(* CODESYS project Copy_of_Sensor_model_new.library
   TcLibraryId: TE140x Module Vendor|Copy_of_Sensor_model_new|0.0.0.3
   Company: TE140x Module Vendor
   Title: Copy_of_Sensor_model_new
   Placeholder: Copy_of_Sensor_model_new
   Version: 0.0.0.3

Project tree, tasks and I/O mapping:
  POUs/
    function block FB_Copy_of_Sensor_model_new [ST]: FB_exit, FB_init, nHResult, eInitExceptionHandling, eUpdateExceptionHandling, nExceptionCnt, stActiveException, bInitialized, bExecute
    TcCOM Wrapper/
      function block FB_Copy_of_Sensor_model_new_TcCOM_InitStruct [ST]: FB_init, FB_afterinit, Reinit, FB_exit, eObjectState, nHResult, ipTcComObject, ipADI, nTaskOid, nTaskPriority, nTaskCycleTimeNs, nTaskPort, nTaskSortOrder, eTraceLevelMax, eModuleCaller, eCallerVerification, eStepSizeAdaptation, eExecutionSequence, bExecute, eAccessLockState, eInitExceptionHandling, eUpdateExceptionHandling, stModuleBuildInfo, bInitialized, nSkippedExecutionCount, stLibraryInfo, stModuleInfo, stModuleGeneratorInfo, stSimulinkModelInfo, eCopy_of_Sensor_model_new_P_Sharing, nCopy_of_Sensor_model_new_P_Definer, stCopy_of_Sensor_model_new_P, fSimulationTime, nCycleCount, nExceptionCount, stExceptionInfo
  DUTs/
    data type ST_FB_Copy_of_Sensor_model_new_FB_Main
    data type ST_FB_Copy_of_Sensor_model_new_FB_exit
    data type ST_FB_Copy_of_Sensor_model_new_FB_init
    data type ST_GetSet_HRESULT
    data type E_FpExcptCtrlSetEx
    data type ST_GetSet_E_FpExcptCtrlSetEx
    data type ST_GetSet_ULINT
    data type ST_ExceptionInfo
    data type ST_GetSet_ST_ExceptionInfo
    data type ST_GetSet_BOOL
    data type T_matrix12xdouble
    data type T_matrix6xdouble
    data type T_matrix3xdouble
    data type E_SimTimeStep
    data type E_SolverMode
    data type E_ssMatrixType
    data type ST_RTWRTModelMethodsInfo
    data type E_slJmBdControl
    data type ST_ssSolverInfo
    data type T_matrix2xdouble
    data type ST_B_MovingAveragepitch_Copy_of_Sensor_model_new_T
    data type ST_B_MovingAveragey_Copy_of_Sensor_model_new_T
    data type ST_B_Copy_of_Sensor_model_new_T
    data type T_ZCSigState
    data type ST_PrevZCX_Copy_of_Sensor_model_new_T
    data type ST_X_Copy_of_Sensor_model_new_T
    data type ST_ExtU_Copy_of_Sensor_model_new_T
    data type ST_ExtY_Copy_of_Sensor_model_new_T
    data type ST_XDis_Copy_of_Sensor_model_new_T
    data type T_matrix2x4xdouble
    data type PLREAL
    data type T_matrix4xdoublepointer
    data type ST_ODE4_IntgData
    data type T_matrix8xuint32
    data type ST_cell_wrap_Copy_of_Sensor_model_new_T
    data type T_matrix9xdouble
    data type ST_dsp_simulink_MovingAverage_Copy_of_Sensor_model_new_T
    data type ST_DW_MovingAveragepitch_Copy_of_Sensor_model_new_T
    data type ST_DW_MovingAveragey_Copy_of_Sensor_model_new_T
    data type ST_DW_Copy_of_Sensor_model_new_T
    data type ST_x08a7a7bbd0e5d629f7d70ceec84eacfe
    data type ST_xf09845edab6c83520d8d57def6d6fe1c
    data type ST_RT_MODEL_Copy_of_Sensor_model_new_T
    data type T_matrix18xdouble
    data type ST_P_Copy_of_Sensor_model_new_T
    data type E_ModuleCaller
    data type E_CallerVerification
    data type E_StepSizeAdaptation
    data type E_ExecutionSequence1
    data type E_FpExcptCtrlSet
    data type ST_TcMatSim_ModuleGeneratorInfo
    data type ST_TcMatSim_SimulinkModelInfo
    data type E_ParameterSharingType
    data type ST_FB_Copy_of_Sensor_model_new_TcCOM_InitStruct
    data type ST_FB_Copy_of_Sensor_model_new_TcCOM_InitStruct_FB_init
    data type ST_FB_Copy_of_Sensor_model_new_TcCOM_InitStruct_FB_afterinit
    data type ST_FB_Copy_of_Sensor_model_new_TcCOM_InitStruct_Reinit
    data type ST_FB_Copy_of_Sensor_model_new_TcCOM_InitStruct_FB_Main
    data type ST_FB_Copy_of_Sensor_model_new_TcCOM_InitStruct_FB_exit
    data type ST_GetSet_TCOM_STATE
    data type ST_GetSet_ITComObject
    data type ST_GetSet_ITcADI
    data type ST_Copy_of_Sensor_model_new_U_T
    data type ST_Copy_of_Sensor_model_new_Y_T
    data type ST_Copy_of_Sensor_model_new_X_T
    data type ST_Copy_of_Sensor_model_new_DW_T
    data type ST_GetSet_OTCID
    data type ST_GetSet_UDINT
    data type ST_GetSet_UINT
    data type ST_GetSet_TcTraceLevel
    data type ST_GetSet_E_ModuleCaller
    data type ST_GetSet_E_CallerVerification
    data type ST_GetSet_E_StepSizeAdaptation
    data type ST_GetSet_E_ExecutionSequence1
    data type ST_GetSet_E_FpExcptCtrlSet
    data type ST_ModuleBuildInfo
    data type ST_GetSet_ST_ModuleBuildInfo
    data type ST_LibraryInfo
    data type ST_GetSet_ST_LibraryInfo
    data type ST_ModuleInfo
    data type ST_GetSet_ST_ModuleInfo
    data type ST_GetSet_ST_TcMatSim_ModuleGeneratorInfo
    data type ST_GetSet_ST_TcMatSim_SimulinkModelInfo
    data type ST_GetSet_E_ParameterSharingType
    data type ST_GetSet_ST_P_Copy_of_Sensor_model_new_T
    data type ST_GetSet_LREAL
  Version/
    global variables Global_Version
*)

// DUTs/ST_FB_Copy_of_Sensor_model_new_FB_Main
{attribute 'TcIecLibraryType'}
{attribute 'hide'}
TYPE ST_FB_Copy_of_Sensor_model_new_FB_Main : 
	STRUCT
		{attribute 'GUID' := '18071995-0000-0000-0000-000000000018'}
		pInst : PVOID;
		result : BOOL;
		 {attribute 'hide'}
		_reserved1 : UINT_24_56;
	END_STRUCT
END_TYPE

// DUTs/ST_FB_Copy_of_Sensor_model_new_FB_exit
{attribute 'TcIecLibraryType'}
{attribute 'hide'}
TYPE ST_FB_Copy_of_Sensor_model_new_FB_exit : 
	STRUCT
		{attribute 'GUID' := '18071995-0000-0000-0000-000000000018'}
		pInst : PVOID;
		bInCopyCode : BOOL;
		result : BOOL;
		 {attribute 'hide'}
		_reserved1 : UINT_16_48;
	END_STRUCT
END_TYPE

// DUTs/ST_FB_Copy_of_Sensor_model_new_FB_init
{attribute 'TcIecLibraryType'}
{attribute 'hide'}
TYPE ST_FB_Copy_of_Sensor_model_new_FB_init : 
	STRUCT
		{attribute 'GUID' := '18071995-0000-0000-0000-000000000018'}
		pInst : PVOID;
		bInitRetains : BOOL;
		bInCopyCode : BOOL;
		result : BOOL;
		 {attribute 'hide'}
		_reserved1 : UINT_8_40;
	END_STRUCT
END_TYPE

// DUTs/ST_GetSet_HRESULT
{attribute 'TcIecLibraryType'}
{attribute 'hide'}
TYPE ST_GetSet_HRESULT : 
	STRUCT
		{attribute 'GUID' := '18071995-0000-0000-0000-000000000018'}
		pInst : PVOID;
		{attribute 'GUID' := '18071995-0000-0000-0000-000000000019'}
		nParam : HRESULT;
		 {attribute 'hide'}
		_reserved1 : UINT_0_32;
	END_STRUCT
END_TYPE

// DUTs/E_FpExcptCtrlSetEx
(* Generated from type 'TcMgSdk.FpExcptCtrlSetEx' *)
{attribute 'TcIecLibraryType'}
TYPE E_FpExcptCtrlSetEx : (
	CallerExceptions:=1, 	(* Use the floating point exception settings provided by the caller *)
	ThrowExceptions:=3, 	(* Enable floating point exceptions on invalid operations and divisions by zero *)
	SuppressExceptions:=13, 	(* Disable floating point exceptions. *)
	LogExceptions:=19, 	(* Log exception information. *)
	LogAndHold:=51, 	(* Log exception information and puase execution of the cyclic code after completion of the actual cycle *)
	LogAndCatch:=83, 	(* Log exception information and immediately terminate execution of the cyclic code. Reinitialization is required to restart. *)
	LogAndDump:=147, 	(* Log exception information, create a dump file with detailed exception information and try to continue execution of the cyclic code *)
	LogHoldAndDump:=179, 	(* Log exception information, create a dump file with detailed exception information and puase execution of the cyclic code after completion of the actual cycle *)
	LogCatchAndDump:=211	(* Log exception information, create a dump file with detailed exception information and immediately terminate execution of the cyclic code. Reinitialization is required to restart. *)
) USINT;
END_TYPE

// DUTs/ST_GetSet_E_FpExcptCtrlSetEx
{attribute 'TcIecLibraryType'}
{attribute 'hide'}
TYPE ST_GetSet_E_FpExcptCtrlSetEx : 
	STRUCT
		{attribute 'GUID' := '18071995-0000-0000-0000-000000000018'}
		pInst : PVOID;
		eParam : E_FpExcptCtrlSetEx;
		 {attribute 'hide'}
		_reserved1 : UINT_24_56;
	END_STRUCT
END_TYPE

// DUTs/ST_GetSet_ULINT
{attribute 'TcIecLibraryType'}
{attribute 'hide'}
TYPE ST_GetSet_ULINT : 
	STRUCT
		{attribute 'GUID' := '18071995-0000-0000-0000-000000000018'}
		pInst : PVOID;
		nParam : ULINT;
	END_STRUCT
END_TYPE

// DUTs/ST_ExceptionInfo
(* Generated from type 'TcMgSdk.ExceptionInfo' *)
{attribute 'TcIecLibraryType'}
TYPE ST_ExceptionInfo : 
	STRUCT
		(* Generated from item 'ExceptionCode' *)
		nExceptionCode : DINT;
		(* Generated from item 'TmxName' *)
		{attribute 'GUID' := '18071995-0000-0000-0000-00010000007F'}
		sTmxName : STRING(127);
		(* Generated from item 'TmxVersion' *)
		nTmxVersion : ARRAY [0..3] OF UDINT;
		(* Generated from item 'InstructionAddr' *)
		nInstructionAddr : UDINT;
		(* Generated from item 'ReturnAddr' *)
		nReturnAddr : ARRAY [0..3] OF UDINT;
		(* Generated from item 'DumpCreated' *)
		bDumpCreated : BOOL;
		 {attribute 'hide'}
		_reserved1 : ARRAY [1..3] OF USINT;
	END_STRUCT
END_TYPE

// DUTs/ST_GetSet_ST_ExceptionInfo
{attribute 'TcIecLibraryType'}
{attribute 'hide'}
TYPE ST_GetSet_ST_ExceptionInfo : 
	STRUCT
		{attribute 'GUID' := '18071995-0000-0000-0000-000000000018'}
		pInst : PVOID;
		stParam : ST_ExceptionInfo;
		 {attribute 'hide'}
		_reserved1 : UINT_0_32;
	END_STRUCT
END_TYPE

// DUTs/ST_GetSet_BOOL
{attribute 'TcIecLibraryType'}
{attribute 'hide'}
TYPE ST_GetSet_BOOL : 
	STRUCT
		{attribute 'GUID' := '18071995-0000-0000-0000-000000000018'}
		pInst : PVOID;
		bParam : BOOL;
		 {attribute 'hide'}
		_reserved1 : UINT_24_56;
	END_STRUCT
END_TYPE

// DUTs/T_matrix12xdouble
(* Generated from type 'matrix12xdouble' *)
{attribute 'TcIecLibraryType'}
TYPE T_matrix12xdouble : ARRAY [0..11] OF LREAL;
END_TYPE

// DUTs/T_matrix6xdouble
(* Generated from type 'matrix6xdouble' *)
{attribute 'TcIecLibraryType'}
TYPE T_matrix6xdouble : ARRAY [0..5] OF LREAL;
END_TYPE

// DUTs/T_matrix3xdouble
(* Generated from type 'matrix3xdouble' *)
{attribute 'TcIecLibraryType'}
TYPE T_matrix3xdouble : ARRAY [0..2] OF LREAL;
END_TYPE

// DUTs/E_SimTimeStep
(* Generated from type 'SimTimeStep' *)
{attribute 'TcIecLibraryType'}
{attribute 'qualified_only' := 'true'}
TYPE E_SimTimeStep : (MINOR_TIME_STEP:=0, MAJOR_TIME_STEP:=1) DINT;
END_TYPE

// DUTs/E_SolverMode
(* Generated from type 'SolverMode' *)
{attribute 'TcIecLibraryType'}
{attribute 'qualified_only' := 'true'}
TYPE E_SolverMode : (SOLVER_MODE_AUTO:=0, SOLVER_MODE_SINGLETASKING:=1, SOLVER_MODE_MULTITASKING:=2) DINT;
END_TYPE

// DUTs/E_ssMatrixType
(* Generated from type 'ssMatrixType' *)
{attribute 'TcIecLibraryType'}
{attribute 'qualified_only' := 'true'}
TYPE E_ssMatrixType : (SS_MATRIX_NONE:=0, SS_MATRIX_CONSTANT:=1, SS_MATRIX_TIMEDEP:=2, SS_MATRIX_STATEDEP:=3) DINT;
END_TYPE

// DUTs/ST_RTWRTModelMethodsInfo
(* Generated from type 'RTWRTModelMethodsInfo' *)
{attribute 'TcIecLibraryType'}
TYPE ST_RTWRTModelMethodsInfo : 
	STRUCT
		(* Generated from item 'rtModelPtr' *)
		{attribute 'GUID' := '18071995-0000-0000-0000-000000000018'}
		prtModelPtr : PVOID;
		(* Generated from item 'rtmInitSizesFcn' *)
		{attribute 'GUID' := '18071995-0000-0000-0000-000000000018'}
		prtmInitSizesFcn : PVOID;
		(* Generated from item 'rtmInitSampTimesFcn' *)
		{attribute 'GUID' := '18071995-0000-0000-0000-000000000018'}
		prtmInitSampTimesFcn : PVOID;
		(* Generated from item 'rtmStartFcn' *)
		{attribute 'GUID' := '18071995-0000-0000-0000-000000000018'}
		prtmStartFcn : PVOID;
		(* Generated from item 'rtmOutputsFcn' *)
		{attribute 'GUID' := '18071995-0000-0000-0000-000000000018'}
		prtmOutputsFcn : PVOID;
		(* Generated from item 'rtmUpdateFcn' *)
		{attribute 'GUID' := '18071995-0000-0000-0000-000000000018'}
		prtmUpdateFcn : PVOID;
		(* Generated from item 'rtmDervisFcn' *)
		{attribute 'GUID' := '18071995-0000-0000-0000-000000000018'}
		prtmDervisFcn : PVOID;
		(* Generated from item 'rtmProjectionFcn' *)
		{attribute 'GUID' := '18071995-0000-0000-0000-000000000018'}
		prtmProjectionFcn : PVOID;
		(* Generated from item 'rtmMassMatrixFcn' *)
		{attribute 'GUID' := '18071995-0000-0000-0000-000000000018'}
		prtmMassMatrixFcn : PVOID;
		(* Generated from item 'rtmForcingFunctionFcn' *)
		{attribute 'GUID' := '18071995-0000-0000-0000-000000000018'}
		prtmForcingFunctionFcn : PVOID;
		(* Generated from item 'rtmTerminateFcn' *)
		{attribute 'GUID' := '18071995-0000-0000-0000-000000000018'}
		prtmTerminateFcn : PVOID;
		(* Generated from item 'rtmDiscreteEventsFcn' *)
		{attribute 'GUID' := '18071995-0000-0000-0000-000000000018'}
		prtmDiscreteEventsFcn : PVOID;
	END_STRUCT
END_TYPE

// DUTs/E_slJmBdControl
(* Generated from type 'slJmBdControl' *)
{attribute 'TcIecLibraryType'}
{attribute 'qualified_only' := 'true'}
TYPE E_slJmBdControl : (SL_JM_BD_AUTO:=0, SL_JM_BD_SPARSE_PERTURBATION:=1, SL_JM_BD_FULL_PERTURBATION:=2, SL_JM_BD_SPARSE_ANALYTICAL:=3, SL_JM_BD_FULL_ANALYTICAL:=4) DINT;
END_TYPE

// DUTs/ST_ssSolverInfo
(* Generated from type 'ssSolverInfo' *)
{attribute 'TcIecLibraryType'}
TYPE ST_ssSolverInfo : 
	STRUCT
		(* Generated from item 'rtModelPtr' *)
		{attribute 'GUID' := '18071995-0000-0000-0000-000000000018'}
		prtModelPtr : PVOID;
		simTimeStepPtr : POINTER TO E_SimTimeStep;
		(* Generated from item 'solverData' *)
		{attribute 'GUID' := '18071995-0000-0000-0000-000000000018'}
		psolverData : PVOID;
		solverName : POINTER TO SINT;
		(* Generated from item 'isVariableStepSolver' *)
		bisVariableStepSolver : BOOL;
		(* Generated from item 'solverNeedsReset' *)
		bsolverNeedsReset : BOOL;
		 {attribute 'hide'}
		_reserved1 : UINT;
		(* Generated from item 'solverMode' *)
		esolverMode : E_SolverMode;
		(* Generated from item 'solverStopTime' *)
		fsolverStopTime : LREAL;
		stepSizePtr : POINTER TO LREAL;
		(* Generated from item 'minStepSize' *)
		fminStepSize : LREAL;
		(* Generated from item 'maxStepSize' *)
		fmaxStepSize : LREAL;
		(* Generated from item 'fixedStepSize' *)
		ffixedStepSize : LREAL;
		(* Generated from item 'solverShapePreserveControl' *)
		nsolverShapePreserveControl : DINT;
		(* Generated from item 'solverMaxConsecutiveMinStep' *)
		nsolverMaxConsecutiveMinStep : DINT;
		(* Generated from item 'maxNumMinSteps' *)
		nmaxNumMinSteps : DINT;
		(* Generated from item 'solverMaxOrder' *)
		nsolverMaxOrder : DINT;
		(* Generated from item 'solverConsecutiveZCsStepRelTol' *)
		fsolverConsecutiveZCsStepRelTol : LREAL;
		(* Generated from item 'solverMaxConsecutiveZCs' *)
		nsolverMaxConsecutiveZCs : DINT;
		(* Generated from item 'solverExtrapolationOrder' *)
		nsolverExtrapolationOrder : DINT;
		(* Generated from item 'solverNumberNewtonIterations' *)
		nsolverNumberNewtonIterations : DINT;
		(* Generated from item 'solverRefineFactor' *)
		nsolverRefineFactor : DINT;
		(* Generated from item 'solverRelTol' *)
		fsolverRelTol : LREAL;
		(* Generated from item 'unused_real_T_1' *)
		funused_real_T_1 : LREAL;
		dXPtr : POINTER TO POINTER TO LREAL;
		tPtr : POINTER TO POINTER TO LREAL;
		numContStatesPtr : POINTER TO DINT;
		contStatesPtr : POINTER TO POINTER TO LREAL;
		numPeriodicContStatesPtr : POINTER TO DINT;
		periodicContStateIndicesPtr : POINTER TO POINTER TO DINT;
		periodicContStateRangesPtr : POINTER TO POINTER TO LREAL;
		zcSignalVector : POINTER TO LREAL;
		zcEventsVector : POINTER TO USINT;
		zcSignalAttrib : POINTER TO USINT;
		(* Generated from item 'zcSignalVectorLength' *)
		nzcSignalVectorLength : DINT;
		 {attribute 'hide'}
		_reserved2 : UINT_0_32;
		reserved : POINTER TO USINT;
		(* Generated from item 'foundContZcEvents' *)
		bfoundContZcEvents : BOOL;
		(* Generated from item 'isAtLeftPostOfContZcEvent' *)
		bisAtLeftPostOfContZcEvent : BOOL;
		(* Generated from item 'isAtRightPostOfContZcEvent' *)
		bisAtRightPostOfContZcEvent : BOOL;
		(* Generated from item 'adaptiveZcDetection' *)
		badaptiveZcDetection : BOOL;
		(* Generated from item 'numZcSignals' *)
		nnumZcSignals : DINT;
		(* Generated from item 'stateProjection' *)
		bstateProjection : BOOL;
		(* Generated from item 'robustResetMethod' *)
		brobustResetMethod : BOOL;
		(* Generated from item 'updateJacobianAtReset' *)
		bupdateJacobianAtReset : BOOL;
		(* Generated from item 'consistencyChecking' *)
		bconsistencyChecking : BOOL;
		(* Generated from item 'massMatrixType' *)
		emassMatrixType : E_ssMatrixType;
		(* Generated from item 'massMatrixNzMax' *)
		nmassMatrixNzMax : DINT;
		 {attribute 'hide'}
		_reserved3 : UINT_0_32;
		massMatrixIr : POINTER TO DINT;
		massMatrixJc : POINTER TO DINT;
		massMatrixPr : POINTER TO LREAL;
		errStatusPtr : POINTER TO POINTER TO SINT;
		modelMethodsPtr : POINTER TO ST_RTWRTModelMethodsInfo;
		(* Generated from item 'zcThreshold' *)
		fzcThreshold : LREAL;
		(* Generated from item 'reserved_1' *)
		nreserved_1 : DINT;
		(* Generated from item 'consecutiveZCsError' *)
		nconsecutiveZCsError : DINT;
		(* Generated from item 'CTOutputIncnstWithState' *)
		bCTOutputIncnstWithState : BOOL;
		(* Generated from item 'isComputingJacobian' *)
		bisComputingJacobian : BOOL;
		 {attribute 'hide'}
		_reserved4 : UINT;
		(* Generated from item 'solverJacobianMethodControl' *)
		esolverJacobianMethodControl : E_slJmBdControl;
		(* Generated from item 'ignoredZcDiagnostic' *)
		nignoredZcDiagnostic : DINT;
		(* Generated from item 'maskedZcDiagnostic' *)
		nmaskedZcDiagnostic : DINT;
		(* Generated from item 'isOutputMethodComputed' *)
		bisOutputMethodComputed : BOOL;
		 {attribute 'hide'}
		_reserved5 : ARRAY [1..3] OF USINT;
		(* Generated from item 'maxZcBracketingIterations' *)
		nmaxZcBracketingIterations : DINT;
		(* Generated from item 'isMinorTimeStepWithModeChange' *)
		bisMinorTimeStepWithModeChange : BOOL;
		 {attribute 'hide'}
		_reserved6 : ARRAY [1..3] OF USINT;
		(* Generated from item 'maxZcPerStep' *)
		nmaxZcPerStep : DINT;
		zcSignalPtr : POINTER TO POINTER TO LREAL;
		(* Generated from item 'contStateDisabledPtr' *)
		bcontStateDisabledPtr : POINTER TO POINTER TO BOOL;
		(* Generated from item 'isContModeFrozen' *)
		bisContModeFrozen : BOOL;
		 {attribute 'hide'}
		_reserved7 : ARRAY [1..7] OF USINT;
	END_STRUCT
END_TYPE

// DUTs/T_matrix2xdouble
(* Generated from type 'matrix2xdouble' *)
{attribute 'TcIecLibraryType'}
TYPE T_matrix2xdouble : ARRAY [0..1] OF LREAL;
END_TYPE

// DUTs/ST_B_MovingAveragepitch_Copy_of_Sensor_model_new_T
(* Generated from type 'B_MovingAveragepitch_Copy_of_Sensor_model_new_T' *)
{attribute 'TcIecLibraryType'}
TYPE ST_B_MovingAveragepitch_Copy_of_Sensor_model_new_T : 
	STRUCT
		(* Generated from item 'MovingAveragepitch' *)
		fMovingAveragepitch : LREAL;
	END_STRUCT
END_TYPE

// DUTs/ST_B_MovingAveragey_Copy_of_Sensor_model_new_T
(* Generated from type 'B_MovingAveragey_Copy_of_Sensor_model_new_T' *)
{attribute 'TcIecLibraryType'}
TYPE ST_B_MovingAveragey_Copy_of_Sensor_model_new_T : 
	STRUCT
		(* Generated from item 'MovingAveragey' *)
		fMovingAveragey : LREAL;
	END_STRUCT
END_TYPE

// DUTs/ST_B_Copy_of_Sensor_model_new_T
(* Generated from type 'B_Copy_of_Sensor_model_new_T' *)
{attribute 'TcIecLibraryType'}
TYPE ST_B_Copy_of_Sensor_model_new_T : 
	STRUCT
		(* Generated from item 'UnitDelay' *)
		fUnitDelay : LREAL;
		(* Generated from item 'UnitDelay1' *)
		fUnitDelay1 : LREAL;
		(* Generated from item 'Convert_to_meters' *)
		aConvert_to_meters : T_matrix12xdouble;
		(* Generated from item 'z' *)
		fz : LREAL;
		(* Generated from item 'roll' *)
		froll : LREAL;
		(* Generated from item 'pitch' *)
		fpitch : LREAL;
		(* Generated from item 'offset_airgaps' *)
		aoffset_airgaps : T_matrix6xdouble;
		(* Generated from item 'corrected_airgaps' *)
		acorrected_airgaps : T_matrix12xdouble;
		(* Generated from item 'n_vertical_sensors_rejected' *)
		fn_vertical_sensors_rejected : LREAL;
		(* Generated from item 'n_lateral_sensors_rejected' *)
		fn_lateral_sensors_rejected : LREAL;
		(* Generated from item 'trigger_vertical_filter' *)
		ftrigger_vertical_filter : LREAL;
		(* Generated from item 'trigger_lateral_filter' *)
		ftrigger_lateral_filter : LREAL;
		(* Generated from item 'y' *)
		fy : LREAL;
		(* Generated from item 'yaw' *)
		fyaw : LREAL;
		(* Generated from item 'offset_airgaps_c' *)
		aoffset_airgaps_c : T_matrix6xdouble;
		(* Generated from item 'airgap_nominal_ems' *)
		aairgap_nominal_ems : T_matrix3xdouble;
		(* Generated from item 'Switch' *)
		aSwitch : T_matrix3xdouble;
		(* Generated from item 'Switch1' *)
		aSwitch1 : T_matrix2xdouble;
		(* Generated from item 'Integrator1' *)
		fIntegrator1 : LREAL;
		(* Generated from item 'RelationalOperator1' *)
		bRelationalOperator1 : BOOL;
		 {attribute 'hide'}
		_reserved1 : ARRAY [1..7] OF USINT;
		(* Generated from item 'MovingAveragez' *)
		stMovingAveragez : ST_B_MovingAveragepitch_Copy_of_Sensor_model_new_T;
		(* Generated from item 'MovingAverageyaw' *)
		stMovingAverageyaw : ST_B_MovingAveragey_Copy_of_Sensor_model_new_T;
		(* Generated from item 'MovingAveragey' *)
		stMovingAveragey : ST_B_MovingAveragey_Copy_of_Sensor_model_new_T;
		(* Generated from item 'MovingAverageroll' *)
		stMovingAverageroll : ST_B_MovingAveragepitch_Copy_of_Sensor_model_new_T;
		(* Generated from item 'MovingAveragepitch' *)
		stMovingAveragepitch : ST_B_MovingAveragepitch_Copy_of_Sensor_model_new_T;
	END_STRUCT
END_TYPE

// DUTs/T_ZCSigState
(* Generated from type 'ZCSigState' *)
{attribute 'TcIecLibraryType'}
TYPE T_ZCSigState : USINT;
END_TYPE

// DUTs/ST_PrevZCX_Copy_of_Sensor_model_new_T
(* Generated from type 'PrevZCX_Copy_of_Sensor_model_new_T' *)
{attribute 'TcIecLibraryType'}
TYPE ST_PrevZCX_Copy_of_Sensor_model_new_T : 
	STRUCT
		(* Generated from item 'Integrator_Reset_ZCE' *)
		nIntegrator_Reset_ZCE : T_ZCSigState;
		(* Generated from item 'Integrator1_Reset_ZCE' *)
		nIntegrator1_Reset_ZCE : T_ZCSigState;
	END_STRUCT
END_TYPE

// DUTs/ST_X_Copy_of_Sensor_model_new_T
(* Generated from type 'X_Copy_of_Sensor_model_new_T' *)
{attribute 'TcIecLibraryType'}
TYPE ST_X_Copy_of_Sensor_model_new_T : 
	STRUCT
		(* Generated from item 'Integrator_CSTATE' *)
		fIntegrator_CSTATE : LREAL;
		(* Generated from item 'Integrator1_CSTATE' *)
		fIntegrator1_CSTATE : LREAL;
	END_STRUCT
END_TYPE

// DUTs/ST_ExtU_Copy_of_Sensor_model_new_T
(* Generated from type 'ExtU_Copy_of_Sensor_model_new_T' *)
{attribute 'TcIecLibraryType'}
TYPE ST_ExtU_Copy_of_Sensor_model_new_T : 
	STRUCT
		(* Generated from item 'Newsensorairgaps' *)
		aNewsensorairgaps : T_matrix12xdouble;
	END_STRUCT
END_TYPE

// DUTs/ST_ExtY_Copy_of_Sensor_model_new_T
(* Generated from type 'ExtY_Copy_of_Sensor_model_new_T' *)
{attribute 'TcIecLibraryType'}
TYPE ST_ExtY_Copy_of_Sensor_model_new_T : 
	STRUCT
		(* Generated from item 'z_filtered' *)
		fz_filtered : LREAL;
		(* Generated from item 'roll_filtered' *)
		froll_filtered : LREAL;
		(* Generated from item 'pitch_filtered' *)
		fpitch_filtered : LREAL;
		(* Generated from item 'y_filtered' *)
		fy_filtered : LREAL;
		(* Generated from item 'yaw_filtered' *)
		fyaw_filtered : LREAL;
		(* Generated from item 'offset_airgaps' *)
		aoffset_airgaps : T_matrix6xdouble;
		(* Generated from item 'offset_airgaps_ems' *)
		aoffset_airgaps_ems : T_matrix6xdouble;
		(* Generated from item 'n_vertical_sensors_rejected' *)
		fn_vertical_sensors_rejected : LREAL;
		(* Generated from item 'n_lateral_sensors_rejected' *)
		fn_lateral_sensors_rejected : LREAL;
		(* Generated from item 'z' *)
		fz : LREAL;
		(* Generated from item 'roll' *)
		froll : LREAL;
		(* Generated from item 'pitch' *)
		fpitch : LREAL;
		(* Generated from item 'y' *)
		fy : LREAL;
		(* Generated from item 'yaw' *)
		fyaw : LREAL;
		(* Generated from item 'airgap_nominal_ems' *)
		aairgap_nominal_ems : T_matrix3xdouble;
	END_STRUCT
END_TYPE

// DUTs/ST_XDis_Copy_of_Sensor_model_new_T
(* Generated from type 'XDis_Copy_of_Sensor_model_new_T' *)
{attribute 'TcIecLibraryType'}
TYPE ST_XDis_Copy_of_Sensor_model_new_T : 
	STRUCT
		(* Generated from item 'Integrator_CSTATE' *)
		bIntegrator_CSTATE : BOOL;
		(* Generated from item 'Integrator1_CSTATE' *)
		bIntegrator1_CSTATE : BOOL;
	END_STRUCT
END_TYPE

// DUTs/T_matrix2x4xdouble
(* Generated from type 'matrix2x4xdouble' *)
{attribute 'TcIecLibraryType'}
TYPE T_matrix2x4xdouble : ARRAY [0..3,0..1] OF LREAL;
END_TYPE

// DUTs/PLREAL
{attribute 'TcIecLibraryType'}
TYPE PLREAL : POINTER TO LREAL;
END_TYPE

// DUTs/T_matrix4xdoublepointer
(* Generated from type 'matrix4xdouble *' *)
{attribute 'TcIecLibraryType'}
{attribute 'BaseTypeGUID' := '2CE33DB5-EBD3-49F7-1FA0-F8105FFA7B54'}
TYPE T_matrix4xdoublepointer : ARRAY [0..3] OF PLREAL;
END_TYPE

// DUTs/ST_ODE4_IntgData
(* Generated from type 'ODE4_IntgData' *)
{attribute 'TcIecLibraryType'}
{attribute 'pack_mode' := '1'}
TYPE ST_ODE4_IntgData : 
	STRUCT
		y : POINTER TO LREAL;
		(* Generated from item 'f' *)
		af : T_matrix4xdoublepointer;
	END_STRUCT
END_TYPE

// DUTs/T_matrix8xuint32
(* Generated from type 'matrix8xuint32' *)
{attribute 'TcIecLibraryType'}
TYPE T_matrix8xuint32 : ARRAY [0..7] OF UDINT;
END_TYPE

// DUTs/ST_cell_wrap_Copy_of_Sensor_model_new_T
(* Generated from type 'cell_wrap_Copy_of_Sensor_model_new_T' *)
{attribute 'TcIecLibraryType'}
TYPE ST_cell_wrap_Copy_of_Sensor_model_new_T : 
	STRUCT
		(* Generated from item 'f1' *)
		af1 : T_matrix8xuint32;
	END_STRUCT
END_TYPE

// DUTs/T_matrix9xdouble
(* Generated from type 'matrix9xdouble' *)
{attribute 'TcIecLibraryType'}
TYPE T_matrix9xdouble : ARRAY [0..8] OF LREAL;
END_TYPE

// DUTs/ST_dsp_simulink_MovingAverage_Copy_of_Sensor_model_new_T
(* Generated from type 'dsp_simulink_MovingAverage_Copy_of_Sensor_model_new_T' *)
{attribute 'TcIecLibraryType'}
TYPE ST_dsp_simulink_MovingAverage_Copy_of_Sensor_model_new_T : 
	STRUCT
		(* Generated from item 'matlabCodegenIsDeleted' *)
		bmatlabCodegenIsDeleted : BOOL;
		 {attribute 'hide'}
		_reserved1 : ARRAY [1..3] OF USINT;
		(* Generated from item 'isInitialized' *)
		nisInitialized : DINT;
		(* Generated from item 'isSetupComplete' *)
		bisSetupComplete : BOOL;
		(* Generated from item 'TunablePropsChanged' *)
		bTunablePropsChanged : BOOL;
		 {attribute 'hide'}
		_reserved2 : UINT;
		(* Generated from item 'inputVarSize' *)
		stinputVarSize : ST_cell_wrap_Copy_of_Sensor_model_new_T;
		(* Generated from item 'NumChannels' *)
		nNumChannels : DINT;
		(* Generated from item 'FrameLength' *)
		nFrameLength : DINT;
		 {attribute 'hide'}
		_reserved3 : UDINT;
		(* Generated from item 'pCumSum' *)
		fpCumSum : LREAL;
		(* Generated from item 'pCumSumRev' *)
		apCumSumRev : T_matrix9xdouble;
		(* Generated from item 'pCumRevIndex' *)
		fpCumRevIndex : LREAL;
		(* Generated from item 'pModValueRev' *)
		fpModValueRev : LREAL;
	END_STRUCT
END_TYPE

// DUTs/ST_DW_MovingAveragepitch_Copy_of_Sensor_model_new_T
(* Generated from type 'DW_MovingAveragepitch_Copy_of_Sensor_model_new_T' *)
{attribute 'TcIecLibraryType'}
TYPE ST_DW_MovingAveragepitch_Copy_of_Sensor_model_new_T : 
	STRUCT
		(* Generated from item 'obj' *)
		stobj : ST_dsp_simulink_MovingAverage_Copy_of_Sensor_model_new_T;
		(* Generated from item 'objisempty' *)
		bobjisempty : BOOL;
		 {attribute 'hide'}
		_reserved1 : ARRAY [1..7] OF USINT;
	END_STRUCT
END_TYPE

// DUTs/ST_DW_MovingAveragey_Copy_of_Sensor_model_new_T
(* Generated from type 'DW_MovingAveragey_Copy_of_Sensor_model_new_T' *)
{attribute 'TcIecLibraryType'}
TYPE ST_DW_MovingAveragey_Copy_of_Sensor_model_new_T : 
	STRUCT
		(* Generated from item 'obj' *)
		stobj : ST_dsp_simulink_MovingAverage_Copy_of_Sensor_model_new_T;
		(* Generated from item 'objisempty' *)
		bobjisempty : BOOL;
		 {attribute 'hide'}
		_reserved1 : ARRAY [1..7] OF USINT;
	END_STRUCT
END_TYPE

// DUTs/ST_DW_Copy_of_Sensor_model_new_T
(* Generated from type 'DW_Copy_of_Sensor_model_new_T' *)
{attribute 'TcIecLibraryType'}
TYPE ST_DW_Copy_of_Sensor_model_new_T : 
	STRUCT
		(* Generated from item 'UnitDelay_DSTATE' *)
		fUnitDelay_DSTATE : LREAL;
		(* Generated from item 'UnitDelay1_DSTATE' *)
		fUnitDelay1_DSTATE : LREAL;
		(* Generated from item 'MovingAveragez' *)
		stMovingAveragez : ST_DW_MovingAveragepitch_Copy_of_Sensor_model_new_T;
		(* Generated from item 'MovingAverageyaw' *)
		stMovingAverageyaw : ST_DW_MovingAveragey_Copy_of_Sensor_model_new_T;
		(* Generated from item 'MovingAveragey' *)
		stMovingAveragey : ST_DW_MovingAveragey_Copy_of_Sensor_model_new_T;
		(* Generated from item 'MovingAverageroll' *)
		stMovingAverageroll : ST_DW_MovingAveragepitch_Copy_of_Sensor_model_new_T;
		(* Generated from item 'MovingAveragepitch' *)
		stMovingAveragepitch : ST_DW_MovingAveragepitch_Copy_of_Sensor_model_new_T;
	END_STRUCT
END_TYPE

// DUTs/ST_x08a7a7bbd0e5d629f7d70ceec84eacfe
(* Generated from type 'x08a7a7bbd0e5d629f7d70ceec84eacfe' *)
{attribute 'TcIecLibraryType'}
TYPE ST_x08a7a7bbd0e5d629f7d70ceec84eacfe : 
	STRUCT
		(* Generated from item 'numContStates' *)
		nnumContStates : DINT;
		(* Generated from item 'numPeriodicContStates' *)
		nnumPeriodicContStates : DINT;
		(* Generated from item 'numSampTimes' *)
		nnumSampTimes : DINT;
	END_STRUCT
END_TYPE

// DUTs/ST_xf09845edab6c83520d8d57def6d6fe1c
(* Generated from type 'xf09845edab6c83520d8d57def6d6fe1c' *)
{attribute 'TcIecLibraryType'}
TYPE ST_xf09845edab6c83520d8d57def6d6fe1c : 
	STRUCT
		(* Generated from item 'clockTick0' *)
		nclockTick0 : UDINT;
		(* Generated from item 'clockTickH0' *)
		nclockTickH0 : UDINT;
		(* Generated from item 'stepSize0' *)
		fstepSize0 : LREAL;
		(* Generated from item 'clockTick1' *)
		nclockTick1 : UDINT;
		(* Generated from item 'clockTickH1' *)
		nclockTickH1 : UDINT;
		(* Generated from item 'tStart' *)
		ftStart : LREAL;
		(* Generated from item 'simTimeStep' *)
		esimTimeStep : E_SimTimeStep;
		(* Generated from item 'stopRequestedFlag' *)
		bstopRequestedFlag : BOOL;
		 {attribute 'hide'}
		_reserved1 : ARRAY [1..3] OF USINT;
		t : POINTER TO LREAL;
		(* Generated from item 'tArray' *)
		atArray : T_matrix2xdouble;
	END_STRUCT
END_TYPE

// DUTs/ST_RT_MODEL_Copy_of_Sensor_model_new_T
(* Generated from type 'RT_MODEL_Copy_of_Sensor_model_new_T' *)
{attribute 'TcIecLibraryType'}
{attribute 'pack_mode' := '1'}
TYPE ST_RT_MODEL_Copy_of_Sensor_model_new_T : 
	STRUCT
		errorStatus : POINTER TO SINT;
		solverInfo : POINTER TO ST_ssSolverInfo;
		blockIO : POINTER TO ST_B_Copy_of_Sensor_model_new_T;
		prevZCSigState : POINTER TO ST_PrevZCX_Copy_of_Sensor_model_new_T;
		contStates : POINTER TO ST_X_Copy_of_Sensor_model_new_T;
		periodicContStateIndices : POINTER TO DINT;
		periodicContStateRanges : POINTER TO LREAL;
		derivs : POINTER TO LREAL;
		inputs : POINTER TO ST_ExtU_Copy_of_Sensor_model_new_T;
		outputs : POINTER TO ST_ExtY_Copy_of_Sensor_model_new_T;
		contStateDisabled : POINTER TO ST_XDis_Copy_of_Sensor_model_new_T;
		(* Generated from item 'zCCacheNeedsReset' *)
		bzCCacheNeedsReset : BOOL;
		(* Generated from item 'derivCacheNeedsReset' *)
		bderivCacheNeedsReset : BOOL;
		(* Generated from item 'CTOutputIncnstWithState' *)
		bCTOutputIncnstWithState : BOOL;
		 {attribute 'hide'}
		_reserved1 : UINT_8_40;
		(* Generated from item 'odeY' *)
		aodeY : T_matrix2xdouble;
		(* Generated from item 'odeF' *)
		aodeF : T_matrix2x4xdouble;
		(* Generated from item 'intgData' *)
		stintgData : ST_ODE4_IntgData;
		dwork : POINTER TO ST_DW_Copy_of_Sensor_model_new_T;
		(* Generated from item 'Sizes' *)
		stSizes : ST_x08a7a7bbd0e5d629f7d70ceec84eacfe;
		 {attribute 'hide'}
		_reserved2 : UDINT;
		(* Generated from item 'Timing' *)
		stTiming : ST_xf09845edab6c83520d8d57def6d6fe1c;
	END_STRUCT
END_TYPE

// DUTs/T_matrix18xdouble
(* Generated from type 'matrix18xdouble' *)
{attribute 'TcIecLibraryType'}
TYPE T_matrix18xdouble : ARRAY [0..17] OF LREAL;
END_TYPE

// DUTs/ST_P_Copy_of_Sensor_model_new_T
(* Generated from type 'P_Copy_of_Sensor_model_new_T' *)
{attribute 'TcIecLibraryType'}
TYPE ST_P_Copy_of_Sensor_model_new_T : 
	STRUCT
		(* Generated from item 'Laser_magnet_offset_EMS' *)
		aLaser_magnet_offset_EMS : T_matrix6xdouble;
		(* Generated from item 'Laser_magnet_offset_HEMS' *)
		aLaser_magnet_offset_HEMS : T_matrix6xdouble;
		(* Generated from item 'coords_lat_sensors' *)
		acoords_lat_sensors : T_matrix12xdouble;
		(* Generated from item 'coords_vert_sensors' *)
		acoords_vert_sensors : T_matrix18xdouble;
		(* Generated from item 'cycle_time' *)
		fcycle_time : LREAL;
		(* Generated from item 'lateral_filter_window_cycles' *)
		flateral_filter_window_cycles : LREAL;
		(* Generated from item 'n_sensors_v' *)
		fn_sensors_v : LREAL;
		(* Generated from item 'vertical_filter_window_cycles' *)
		fvertical_filter_window_cycles : LREAL;
		(* Generated from item 'z_com' *)
		fz_com : LREAL;
		(* Generated from item 'UnitDelay_InitialCondition' *)
		fUnitDelay_InitialCondition : LREAL;
		(* Generated from item 'UnitDelay1_InitialCondition' *)
		fUnitDelay1_InitialCondition : LREAL;
		(* Generated from item 'Convert_to_meters_Gain' *)
		fConvert_to_meters_Gain : LREAL;
		(* Generated from item 'Integrator_IC' *)
		fIntegrator_IC : LREAL;
		(* Generated from item 'Integrator1_IC' *)
		fIntegrator1_IC : LREAL;
		(* Generated from item 'Constant_Value' *)
		fConstant_Value : LREAL;
	END_STRUCT
END_TYPE

// DUTs/E_ModuleCaller
(* Generated from type 'TcMgSdk.ModuleCaller' *)
{attribute 'TcIecLibraryType'}
TYPE E_ModuleCaller : (
	CyclicTask:=0, 	(* Add to the specified cyclic caller tasks. *)
	Module:=1	(* Don't add to cyclic callers. The module can be called from other TwinCAT modules (e. g. a PLC). *)
) DINT;
END_TYPE

// DUTs/E_CallerVerification
(* Generated from type 'TcMgSdk.CallerVerification' *)
{attribute 'TcIecLibraryType'}
TYPE E_CallerVerification : (
	Default:=0, 	(* Verify the caller task only if the "ModuleCaller" parameter is set to "Module" but not when added to cyclic caller tasks. *)
	Always:=1, 	(* Always verify the caller context to prevent concurrent execution of model code and corresponding DataArea mappings. *)
	Never:=2	(* Skip caller verification to reduce execution times. *)
) DINT;
END_TYPE

// DUTs/E_StepSizeAdaptation
(* Generated from type 'TcMgSdk.StepSizeAdaptation' *)
{attribute 'TcIecLibraryType'}
TYPE E_StepSizeAdaptation : (
	RequireMatchingTaskCycleTime:=0, 	(* Don't accept task cycle times other than the Simulink step sizes. *)
	UseTaskCycleTime:=1, 	(* Adapt the Smulink step sizes to the task cycle times. *)
	UseModelStepSize:=2	(* Keep the Smulink step sizes, independent of the callers cycle time. *)
) DINT;
END_TYPE

// DUTs/E_ExecutionSequence1
(* Generated from type 'TcMgSdk.ExecutionSequence1' *)
{attribute 'TcIecLibraryType'}
TYPE E_ExecutionSequence1 : (
	UpdateBeforeOutputMapping:=0, 	(* Input mapping -> State and output update -> Output mapping -> ADS processing *)
	IoAtTaskBegin:=1	(* Input mapping -> Code execution -> Output update -> ADS processing *)
) DINT;
END_TYPE

// DUTs/E_FpExcptCtrlSet
(* Generated from type 'TcMgSdk.FpExcptCtrlSet' *)
{attribute 'TcIecLibraryType'}
TYPE E_FpExcptCtrlSet : (
	CallerExceptions:=1, 	(* Use the floating point exception settings provided by the caller *)
	ThrowExceptions:=3, 	(* Enable floating point exceptions on invalid operations and divisions by zero *)
	SuppressExceptions:=5	(* Disable floating point exceptions. *)
) USINT;
END_TYPE

// DUTs/ST_TcMatSim_ModuleGeneratorInfo
(* Generated from type 'TcMatSim.ModuleGeneratorInfo' *)
{attribute 'TcIecLibraryType'}
TYPE ST_TcMatSim_ModuleGeneratorInfo : 
	STRUCT
		(* Generated from item 'MatlabVersion' *)
		nMatlabVersion : ARRAY [0..3] OF UDINT;
		(* Generated from item 'TE140xVersion' *)
		nTE140xVersion : ARRAY [0..3] OF UDINT;
	END_STRUCT
END_TYPE

// DUTs/ST_TcMatSim_SimulinkModelInfo
(* Generated from type 'TcMatSim.SimulinkModelInfo' *)
{attribute 'TcIecLibraryType'}
TYPE ST_TcMatSim_SimulinkModelInfo : 
	STRUCT
		(* Generated from item 'ModelName' *)
		{attribute 'GUID' := '18071995-0000-0000-0000-00010000007F'}
		sModelName : STRING(127);
		(* Generated from item 'SimulinkVersion' *)
		nSimulinkVersion : ARRAY [0..3] OF UDINT;
		(* Generated from item 'ModelVersion' *)
		nModelVersion : ARRAY [0..3] OF UDINT;
		(* Generated from item 'ModelChecksum' *)
		nModelChecksum : ARRAY [0..3] OF UDINT;
	END_STRUCT
END_TYPE

// DUTs/E_ParameterSharingType
(* Generated from type 'ParameterSharingType' *)
{attribute 'TcIecLibraryType'}
TYPE E_ParameterSharingType : (
	Define:=0, 	(* This module instance defines the parameter values for all further instances of this module class. Exactly one instance of this module class must use this option. *)
	Inherit:=1	(* This module instance inherits the parameter values from the instance of this module class configured to "Define" the parameter values. Model parameters configured at this instsance are ignored. *)
) DINT;
END_TYPE

// DUTs/ST_FB_Copy_of_Sensor_model_new_TcCOM_InitStruct
{attribute 'TcIecLibraryType'}
TYPE ST_FB_Copy_of_Sensor_model_new_TcCOM_InitStruct : 
	STRUCT
		{attribute 'GUID' := '18071995-0000-0000-0000-000000000061'}
		eObjState : TCOM_STATE := TCOM_STATE.TCOM_STATE_OP;
		{attribute 'GUID' := '18071995-0000-0000-0000-00010000007F'}
		sObjName : STRING(127);
		{attribute 'GUID' := '18071995-0000-0000-0000-00000000000F'}
		nOid : OTCID := 4294967295;
		{attribute 'GUID' := '18071995-0000-0000-0000-00000000000F'}
		nTaskOid : OTCID;
		nTaskSortOrder : UDINT;
		{attribute 'GUID' := '8007AE3B-86BB-40F2-B385-EF87FCC239A4'}
		eTraceLevelMax : TcTraceLevel := TcTraceLevel.tlInfo;
		eModuleCaller : E_ModuleCaller := E_ModuleCaller.CyclicTask;
		eCallerVerification : E_CallerVerification := E_CallerVerification.Default;
		eStepSizeAdaptation : E_StepSizeAdaptation := E_StepSizeAdaptation.RequireMatchingTaskCycleTime;
		eExecutionSequence : E_ExecutionSequence1 := E_ExecutionSequence1.UpdateBeforeOutputMapping;
		bExecute : BOOL := TRUE;
		 {attribute 'hide'}
		_reserved1 : ARRAY [1..3] OF USINT;
		{attribute 'GUID' := '18071995-0000-0000-0000-000000000061'}
		eAccessLockState : TCOM_STATE := TCOM_STATE.TCOM_STATE_OP;
		eInitExceptionHandling : E_FpExcptCtrlSet := E_FpExcptCtrlSet.CallerExceptions;
		eUpdateExceptionHandling : E_FpExcptCtrlSetEx := E_FpExcptCtrlSetEx.CallerExceptions;
		 {attribute 'hide'}
		_reserved2 : UINT;
		stModuleGeneratorInfo : ST_TcMatSim_ModuleGeneratorInfo;
		stSimulinkModelInfo : ST_TcMatSim_SimulinkModelInfo;
		eCopy_of_Sensor_model_new_P_Sharing : E_ParameterSharingType := E_ParameterSharingType.Define;
		 {attribute 'hide'}
		_reserved3 : UDINT;
		stCopy_of_Sensor_model_new_P : ST_P_Copy_of_Sensor_model_new_T := (aLaser_magnet_offset_EMS := [0.028731,0.0309094,0.02935319,0.02708477,0.02997081,0.02840083], aLaser_magnet_offset_HEMS := [0.01781551,0.01975221,0.02068667,0.02088624,0.01921297,0.0207209], acoords_lat_sensors := [0.8879802,0.0045598,0.8879802,0.0045598,0.0147302,0.0045598,0.0147302,0.0045598,-0.8585198,0.0045598,-0.8585198,0.0045598], acoords_vert_sensors := [0.8879802,0.3635598,0.0,0.8879802,-0.3544402,0.0,0.1997302,0.3785598,0.0,-0.1702698,-0.3694402,0.0,-0.8585198,0.3635598,0.0,-0.8585198,-0.3544402,0.0], fcycle_time := 0.0015, flateral_filter_window_cycles := 10, fn_sensors_v := 6, fvertical_filter_window_cycles := 10, fz_com := 0.5706599999999999, fUnitDelay_InitialCondition := 0, fUnitDelay1_InitialCondition := 0, fConvert_to_meters_Gain := 0.001, fIntegrator_IC := 0, fIntegrator1_IC := 0, fConstant_Value := 1);
	END_STRUCT
END_TYPE

// DUTs/ST_FB_Copy_of_Sensor_model_new_TcCOM_InitStruct_FB_init
{attribute 'TcIecLibraryType'}
{attribute 'hide'}
TYPE ST_FB_Copy_of_Sensor_model_new_TcCOM_InitStruct_FB_init : 
	STRUCT
		{attribute 'GUID' := '18071995-0000-0000-0000-000000000018'}
		pInst : PVOID;
		bInitRetains : BOOL;
		bInCopyCode : BOOL;
		 {attribute 'hide'}
		_reserved1 : UINT_16_48;
		stInit : REFERENCE TO ST_FB_Copy_of_Sensor_model_new_TcCOM_InitStruct;
		result : BOOL;
		 {attribute 'hide'}
		_reserved2 : UINT_24_56;
	END_STRUCT
END_TYPE

// DUTs/ST_FB_Copy_of_Sensor_model_new_TcCOM_InitStruct_FB_afterinit
{attribute 'TcIecLibraryType'}
{attribute 'hide'}
TYPE ST_FB_Copy_of_Sensor_model_new_TcCOM_InitStruct_FB_afterinit : 
	STRUCT
		{attribute 'GUID' := '18071995-0000-0000-0000-000000000018'}
		pInst : PVOID;
		result : BOOL;
		 {attribute 'hide'}
		_reserved1 : UINT_24_56;
	END_STRUCT
END_TYPE

// DUTs/ST_FB_Copy_of_Sensor_model_new_TcCOM_InitStruct_Reinit
{attribute 'TcIecLibraryType'}
{attribute 'hide'}
TYPE ST_FB_Copy_of_Sensor_model_new_TcCOM_InitStruct_Reinit : 
	STRUCT
		{attribute 'GUID' := '18071995-0000-0000-0000-000000000018'}
		pInst : PVOID;
		stReInit : ST_FB_Copy_of_Sensor_model_new_TcCOM_InitStruct;
		result : BOOL;
		 {attribute 'hide'}
		_reserved1 : ARRAY [1..7] OF USINT;
	END_STRUCT
END_TYPE

// DUTs/ST_FB_Copy_of_Sensor_model_new_TcCOM_InitStruct_FB_Main
{attribute 'TcIecLibraryType'}
{attribute 'hide'}
TYPE ST_FB_Copy_of_Sensor_model_new_TcCOM_InitStruct_FB_Main : 
	STRUCT
		{attribute 'GUID' := '18071995-0000-0000-0000-000000000018'}
		pInst : PVOID;
		result : BOOL;
		 {attribute 'hide'}
		_reserved1 : UINT_24_56;
	END_STRUCT
END_TYPE

// DUTs/ST_FB_Copy_of_Sensor_model_new_TcCOM_InitStruct_FB_exit
{attribute 'TcIecLibraryType'}
{attribute 'hide'}
TYPE ST_FB_Copy_of_Sensor_model_new_TcCOM_InitStruct_FB_exit : 
	STRUCT
		{attribute 'GUID' := '18071995-0000-0000-0000-000000000018'}
		pInst : PVOID;
		bInCopyCode : BOOL;
		result : BOOL;
		 {attribute 'hide'}
		_reserved1 : UINT_16_48;
	END_STRUCT
END_TYPE

// DUTs/ST_GetSet_TCOM_STATE
{attribute 'TcIecLibraryType'}
{attribute 'hide'}
TYPE ST_GetSet_TCOM_STATE : 
	STRUCT
		{attribute 'GUID' := '18071995-0000-0000-0000-000000000018'}
		pInst : PVOID;
		{attribute 'GUID' := '18071995-0000-0000-0000-000000000061'}
		eParam : TCOM_STATE;
		 {attribute 'hide'}
		_reserved1 : UINT_0_32;
	END_STRUCT
END_TYPE

// DUTs/ST_GetSet_ITComObject
{attribute 'TcIecLibraryType'}
{attribute 'hide'}
TYPE ST_GetSet_ITComObject : 
	STRUCT
		{attribute 'GUID' := '18071995-0000-0000-0000-000000000018'}
		pInst : PVOID;
		{attribute 'GUID' := '00000012-0000-0000-E000-000000000064'}
		ipParam : ITComObject;
	END_STRUCT
END_TYPE

// DUTs/ST_GetSet_ITcADI
{attribute 'TcIecLibraryType'}
{attribute 'hide'}
TYPE ST_GetSet_ITcADI : 
	STRUCT
		{attribute 'GUID' := '18071995-0000-0000-0000-000000000018'}
		pInst : PVOID;
		{attribute 'GUID' := '03000012-0000-0000-E000-000000000064'}
		ipParam : ITcADI;
	END_STRUCT
END_TYPE

// DUTs/ST_Copy_of_Sensor_model_new_U_T
(* Generated from type 'Copy_of_Sensor_model_new_U_T' *)
{attribute 'TcIecLibraryType'}
TYPE ST_Copy_of_Sensor_model_new_U_T : 
	STRUCT
		(* Generated from item 'Newsensorairgaps' *)
		aNewsensorairgaps : T_matrix12xdouble;
	END_STRUCT
END_TYPE

// DUTs/ST_Copy_of_Sensor_model_new_Y_T
(* Generated from type 'Copy_of_Sensor_model_new_Y_T' *)
{attribute 'TcIecLibraryType'}
TYPE ST_Copy_of_Sensor_model_new_Y_T : 
	STRUCT
		(* Generated from item 'z_filtered' *)
		fz_filtered : LREAL;
		(* Generated from item 'roll_filtered' *)
		froll_filtered : LREAL;
		(* Generated from item 'pitch_filtered' *)
		fpitch_filtered : LREAL;
		(* Generated from item 'y_filtered' *)
		fy_filtered : LREAL;
		(* Generated from item 'yaw_filtered' *)
		fyaw_filtered : LREAL;
		(* Generated from item 'offset_airgaps' *)
		aoffset_airgaps : T_matrix6xdouble;
		(* Generated from item 'offset_airgaps_ems' *)
		aoffset_airgaps_ems : T_matrix6xdouble;
		(* Generated from item 'n_vertical_sensors_rejected' *)
		fn_vertical_sensors_rejected : LREAL;
		(* Generated from item 'n_lateral_sensors_rejected' *)
		fn_lateral_sensors_rejected : LREAL;
		(* Generated from item 'z' *)
		fz : LREAL;
		(* Generated from item 'roll' *)
		froll : LREAL;
		(* Generated from item 'pitch' *)
		fpitch : LREAL;
		(* Generated from item 'y' *)
		fy : LREAL;
		(* Generated from item 'yaw' *)
		fyaw : LREAL;
		(* Generated from item 'airgap_nominal_ems' *)
		aairgap_nominal_ems : T_matrix3xdouble;
	END_STRUCT
END_TYPE

// DUTs/ST_Copy_of_Sensor_model_new_X_T
(* Generated from type 'Copy_of_Sensor_model_new_X_T' *)
{attribute 'TcIecLibraryType'}
TYPE ST_Copy_of_Sensor_model_new_X_T : 
	STRUCT
		(* Generated from item 'Integrator_CSTATE' *)
		fIntegrator_CSTATE : LREAL;
		(* Generated from item 'Integrator1_CSTATE' *)
		fIntegrator1_CSTATE : LREAL;
	END_STRUCT
END_TYPE

// DUTs/ST_Copy_of_Sensor_model_new_DW_T
(* Generated from type 'Copy_of_Sensor_model_new_DW_T' *)
{attribute 'TcIecLibraryType'}
TYPE ST_Copy_of_Sensor_model_new_DW_T : 
	STRUCT
		(* Generated from item 'UnitDelay_DSTATE' *)
		fUnitDelay_DSTATE : LREAL;
		(* Generated from item 'UnitDelay1_DSTATE' *)
		fUnitDelay1_DSTATE : LREAL;
		(* Generated from item 'MovingAveragez' *)
		stMovingAveragez : ST_DW_MovingAveragepitch_Copy_of_Sensor_model_new_T;
		(* Generated from item 'MovingAverageyaw' *)
		stMovingAverageyaw : ST_DW_MovingAveragey_Copy_of_Sensor_model_new_T;
		(* Generated from item 'MovingAveragey' *)
		stMovingAveragey : ST_DW_MovingAveragey_Copy_of_Sensor_model_new_T;
		(* Generated from item 'MovingAverageroll' *)
		stMovingAverageroll : ST_DW_MovingAveragepitch_Copy_of_Sensor_model_new_T;
		(* Generated from item 'MovingAveragepitch' *)
		stMovingAveragepitch : ST_DW_MovingAveragepitch_Copy_of_Sensor_model_new_T;
	END_STRUCT
END_TYPE

// DUTs/ST_GetSet_OTCID
{attribute 'TcIecLibraryType'}
{attribute 'hide'}
TYPE ST_GetSet_OTCID : 
	STRUCT
		{attribute 'GUID' := '18071995-0000-0000-0000-000000000018'}
		pInst : PVOID;
		{attribute 'GUID' := '18071995-0000-0000-0000-00000000000F'}
		nParam : OTCID;
		 {attribute 'hide'}
		_reserved1 : UINT_0_32;
	END_STRUCT
END_TYPE

// DUTs/ST_GetSet_UDINT
{attribute 'TcIecLibraryType'}
{attribute 'hide'}
TYPE ST_GetSet_UDINT : 
	STRUCT
		{attribute 'GUID' := '18071995-0000-0000-0000-000000000018'}
		pInst : PVOID;
		nParam : UDINT;
		 {attribute 'hide'}
		_reserved1 : UINT_0_32;
	END_STRUCT
END_TYPE

// DUTs/ST_GetSet_UINT
{attribute 'TcIecLibraryType'}
{attribute 'hide'}
TYPE ST_GetSet_UINT : 
	STRUCT
		{attribute 'GUID' := '18071995-0000-0000-0000-000000000018'}
		pInst : PVOID;
		nParam : UINT;
		 {attribute 'hide'}
		_reserved1 : UINT_16_48;
	END_STRUCT
END_TYPE

// DUTs/ST_GetSet_TcTraceLevel
{attribute 'TcIecLibraryType'}
{attribute 'hide'}
TYPE ST_GetSet_TcTraceLevel : 
	STRUCT
		{attribute 'GUID' := '18071995-0000-0000-0000-000000000018'}
		pInst : PVOID;
		{attribute 'GUID' := '8007AE3B-86BB-40F2-B385-EF87FCC239A4'}
		eParam : TcTraceLevel;
		 {attribute 'hide'}
		_reserved1 : UINT_0_32;
	END_STRUCT
END_TYPE

// DUTs/ST_GetSet_E_ModuleCaller
{attribute 'TcIecLibraryType'}
{attribute 'hide'}
TYPE ST_GetSet_E_ModuleCaller : 
	STRUCT
		{attribute 'GUID' := '18071995-0000-0000-0000-000000000018'}
		pInst : PVOID;
		eParam : E_ModuleCaller;
		 {attribute 'hide'}
		_reserved1 : UINT_0_32;
	END_STRUCT
END_TYPE

// DUTs/ST_GetSet_E_CallerVerification
{attribute 'TcIecLibraryType'}
{attribute 'hide'}
TYPE ST_GetSet_E_CallerVerification : 
	STRUCT
		{attribute 'GUID' := '18071995-0000-0000-0000-000000000018'}
		pInst : PVOID;
		eParam : E_CallerVerification;
		 {attribute 'hide'}
		_reserved1 : UINT_0_32;
	END_STRUCT
END_TYPE

// DUTs/ST_GetSet_E_StepSizeAdaptation
{attribute 'TcIecLibraryType'}
{attribute 'hide'}
TYPE ST_GetSet_E_StepSizeAdaptation : 
	STRUCT
		{attribute 'GUID' := '18071995-0000-0000-0000-000000000018'}
		pInst : PVOID;
		eParam : E_StepSizeAdaptation;
		 {attribute 'hide'}
		_reserved1 : UINT_0_32;
	END_STRUCT
END_TYPE

// DUTs/ST_GetSet_E_ExecutionSequence1
{attribute 'TcIecLibraryType'}
{attribute 'hide'}
TYPE ST_GetSet_E_ExecutionSequence1 : 
	STRUCT
		{attribute 'GUID' := '18071995-0000-0000-0000-000000000018'}
		pInst : PVOID;
		eParam : E_ExecutionSequence1;
		 {attribute 'hide'}
		_reserved1 : UINT_0_32;
	END_STRUCT
END_TYPE

// DUTs/ST_GetSet_E_FpExcptCtrlSet
{attribute 'TcIecLibraryType'}
{attribute 'hide'}
TYPE ST_GetSet_E_FpExcptCtrlSet : 
	STRUCT
		{attribute 'GUID' := '18071995-0000-0000-0000-000000000018'}
		pInst : PVOID;
		eParam : E_FpExcptCtrlSet;
		 {attribute 'hide'}
		_reserved1 : UINT_24_56;
	END_STRUCT
END_TYPE

// DUTs/ST_ModuleBuildInfo
(* Generated from type 'TcMgSdk.ModuleBuildInfo' *)
{attribute 'TcIecLibraryType'}
TYPE ST_ModuleBuildInfo : 
	STRUCT
		(* Generated from item 'TcBuild' *)
		nTcBuild : UDINT;
		(* Generated from item 'TcRevision' *)
		nTcRevision : UDINT;
		(* Generated from item 'Debug' *)
		bDebug : BOOL;
		 {attribute 'hide'}
		_reserved1 : ARRAY [1..3] OF USINT;
	END_STRUCT
END_TYPE

// DUTs/ST_GetSet_ST_ModuleBuildInfo
{attribute 'TcIecLibraryType'}
{attribute 'hide'}
TYPE ST_GetSet_ST_ModuleBuildInfo : 
	STRUCT
		{attribute 'GUID' := '18071995-0000-0000-0000-000000000018'}
		pInst : PVOID;
		stParam : ST_ModuleBuildInfo;
		 {attribute 'hide'}
		_reserved1 : UINT_0_32;
	END_STRUCT
END_TYPE

// DUTs/ST_LibraryInfo
(* Generated from type 'TcMgSdk.LibraryInfo' *)
{attribute 'TcIecLibraryType'}
TYPE ST_LibraryInfo : 
	STRUCT
		(* Generated from item 'FileVersion' *)
		nFileVersion : ARRAY [0..3] OF UDINT;
		(* Generated from item 'ProductVersion' *)
		nProductVersion : ARRAY [0..3] OF UDINT;
		(* Generated from item 'VendorName' *)
		{attribute 'GUID' := '18071995-0000-0000-0000-00010000007F'}
		sVendorName : STRING(127);
		(* Generated from item 'LibraryName' *)
		{attribute 'GUID' := '18071995-0000-0000-0000-00010000007F'}
		sLibraryName : STRING(127);
		(* Generated from item 'LibraryVersion' *)
		nLibraryVersion : ARRAY [0..3] OF UDINT;
		(* Generated from item 'LibraryId' *)
		{attribute 'GUID' := '18071995-0000-0000-0000-00010000007F'}
		sLibraryId : STRING(127);
		(* Generated from item 'LibraryGUID' *)
		{attribute 'GUID' := '18071995-0000-0000-0000-000000000024'}
		nLibraryGUID : CLSID;
		(* Generated from item 'TcSdkVersion' *)
		nTcSdkVersion : ARRAY [0..3] OF UDINT;
		(* Generated from item 'Compiler' *)
		{attribute 'GUID' := '18071995-0000-0000-0000-00010000007F'}
		sCompiler : STRING(127);
		(* Generated from item 'Debug' *)
		bDebug : BOOL;
		 {attribute 'hide'}
		_reserved1 : ARRAY [1..7] OF USINT;
	END_STRUCT
END_TYPE

// DUTs/ST_GetSet_ST_LibraryInfo
{attribute 'TcIecLibraryType'}
{attribute 'hide'}
TYPE ST_GetSet_ST_LibraryInfo : 
	STRUCT
		{attribute 'GUID' := '18071995-0000-0000-0000-000000000018'}
		pInst : PVOID;
		stParam : ST_LibraryInfo;
	END_STRUCT
END_TYPE

// DUTs/ST_ModuleInfo
(* Generated from type 'TcMgSdk.ModuleInfo' *)
{attribute 'TcIecLibraryType'}
TYPE ST_ModuleInfo : 
	STRUCT
		(* Generated from item 'ClassName' *)
		{attribute 'GUID' := '18071995-0000-0000-0000-00010000007F'}
		sClassName : STRING(127);
		(* Generated from item 'CommonClassId' *)
		{attribute 'GUID' := '18071995-0000-0000-0000-000000000024'}
		nCommonClassId : CLSID;
		(* Generated from item 'VersionClassId' *)
		{attribute 'GUID' := '18071995-0000-0000-0000-000000000024'}
		nVersionClassId : CLSID;
	END_STRUCT
END_TYPE

// DUTs/ST_GetSet_ST_ModuleInfo
{attribute 'TcIecLibraryType'}
{attribute 'hide'}
TYPE ST_GetSet_ST_ModuleInfo : 
	STRUCT
		{attribute 'GUID' := '18071995-0000-0000-0000-000000000018'}
		pInst : PVOID;
		stParam : ST_ModuleInfo;
	END_STRUCT
END_TYPE

// DUTs/ST_GetSet_ST_TcMatSim_ModuleGeneratorInfo
{attribute 'TcIecLibraryType'}
{attribute 'hide'}
TYPE ST_GetSet_ST_TcMatSim_ModuleGeneratorInfo : 
	STRUCT
		{attribute 'GUID' := '18071995-0000-0000-0000-000000000018'}
		pInst : PVOID;
		stParam : ST_TcMatSim_ModuleGeneratorInfo;
	END_STRUCT
END_TYPE

// DUTs/ST_GetSet_ST_TcMatSim_SimulinkModelInfo
{attribute 'TcIecLibraryType'}
{attribute 'hide'}
TYPE ST_GetSet_ST_TcMatSim_SimulinkModelInfo : 
	STRUCT
		{attribute 'GUID' := '18071995-0000-0000-0000-000000000018'}
		pInst : PVOID;
		stParam : ST_TcMatSim_SimulinkModelInfo;
	END_STRUCT
END_TYPE

// DUTs/ST_GetSet_E_ParameterSharingType
{attribute 'TcIecLibraryType'}
{attribute 'hide'}
TYPE ST_GetSet_E_ParameterSharingType : 
	STRUCT
		{attribute 'GUID' := '18071995-0000-0000-0000-000000000018'}
		pInst : PVOID;
		eParam : E_ParameterSharingType;
		 {attribute 'hide'}
		_reserved1 : UINT_0_32;
	END_STRUCT
END_TYPE

// DUTs/ST_GetSet_ST_P_Copy_of_Sensor_model_new_T
{attribute 'TcIecLibraryType'}
{attribute 'hide'}
TYPE ST_GetSet_ST_P_Copy_of_Sensor_model_new_T : 
	STRUCT
		{attribute 'GUID' := '18071995-0000-0000-0000-000000000018'}
		pInst : PVOID;
		stParam : ST_P_Copy_of_Sensor_model_new_T;
	END_STRUCT
END_TYPE

// DUTs/ST_GetSet_LREAL
{attribute 'TcIecLibraryType'}
{attribute 'hide'}
TYPE ST_GetSet_LREAL : 
	STRUCT
		{attribute 'GUID' := '18071995-0000-0000-0000-000000000018'}
		pInst : PVOID;
		fParam : LREAL;
	END_STRUCT
END_TYPE

// Version/Global_Version
{attribute 'TcGenerated'}
// This function has been automatically generated from the project information.
VAR_GLOBAL CONSTANT
	{attribute 'const_non_replaced'}
	{attribute 'linkalways'}
	stLibVersion_Copy_of_Sensor_model_new : ST_LibVersion := (iMajor := 0, iMinor := 0, iBuild := 0, iRevision := 3, nFlags := 0, sVersion := '0.0.0.3');
	{attribute 'const_non_replaced'}
	{attribute 'linkalways'}
	sLibraryId_Copy_of_Sensor_model_new : String := 'TE140x Module Vendor|Copy_of_Sensor_model_new|0.0.0.3';
END_VAR

// POUs/FB_Copy_of_Sensor_model_new

{attribute 'c++_compatible'}
{attribute 'external_name' := 'FB_Copy_of_Sensor_model_new_GUID_8246615A_7393_339B_DD7E_2FC876113668'}
{attribute 'TcIecLibraryType'}
{attribute 'reflection'}
FUNCTION_BLOCK FB_Copy_of_Sensor_model_new
VAR
	{attribute 'hide'}
	{attribute 'no_copy'}
	{attribute 'GUID' := '18071995-0000-0000-0000-000000000018'}
	m_pData : PVOID;
	{attribute 'TcInitSymbol'}
	{attribute 'GUID' := '8007AE3B-86BB-40F2-B385-EF87FCC239A4'}
	eTraceLevelMax : TcTraceLevel := TcTraceLevel.tlInfo;
	 {attribute 'hide'}
	_reserved1 : UDINT;
	{attribute 'hide'}
	{attribute 'instance-path'}
	{attribute 'noinit'}
	{attribute 'GUID' := '18071995-0000-0000-0000-0001000000FF'}
	sInstancePath : STRING(255);
	{attribute 'hide'}
	{attribute 'noinit'}
	{attribute 'GUID' := '18071995-0000-0000-0000-000000000019'}
	m_HResultLog : HRESULT;
	{attribute 'hide'}
	{attribute 'noinit'}
	{attribute 'GUID' := '18071995-0000-0000-0000-000000000019'}
	m_HResult : HRESULT;
	 {attribute 'hide'}
	_reserved2 : ARRAY [1..184] OF USINT;
	{attribute 'hide'}
	{attribute 'no_copy'}
	m_ExtModeData : ULINT;
END_VAR
VAR_INPUT
	(* Generated from item 'Newsensorairgaps' *)
	aNewsensorairgaps : T_matrix12xdouble;
END_VAR
VAR_OUTPUT
	(* Generated from item 'z_filtered' *)
	fz_filtered : LREAL;
	(* Generated from item 'roll_filtered' *)
	froll_filtered : LREAL;
	(* Generated from item 'pitch_filtered' *)
	fpitch_filtered : LREAL;
	(* Generated from item 'y_filtered' *)
	fy_filtered : LREAL;
	(* Generated from item 'yaw_filtered' *)
	fyaw_filtered : LREAL;
	(* Generated from item 'offset_airgaps' *)
	aoffset_airgaps : T_matrix6xdouble;
	(* Generated from item 'offset_airgaps_ems' *)
	aoffset_airgaps_ems : T_matrix6xdouble;
	(* Generated from item 'n_vertical_sensors_rejected' *)
	fn_vertical_sensors_rejected : LREAL;
	(* Generated from item 'n_lateral_sensors_rejected' *)
	fn_lateral_sensors_rejected : LREAL;
	(* Generated from item 'z' *)
	fz : LREAL;
	(* Generated from item 'roll' *)
	froll : LREAL;
	(* Generated from item 'pitch' *)
	fpitch : LREAL;
	(* Generated from item 'y' *)
	fy : LREAL;
	(* Generated from item 'yaw' *)
	fyaw : LREAL;
	(* Generated from item 'airgap_nominal_ems' *)
	aairgap_nominal_ems : T_matrix3xdouble;
END_VAR
VAR
	{attribute 'no_copy'}
	PCopy_of_Sensor_model_new_M : POINTER TO ST_RT_MODEL_Copy_of_Sensor_model_new_T;
END_VAR

{attribute 'TcTypeSystem'}

METHOD FB_exit : BOOL
VAR_INPUT
	bInCopyCode : BOOL;
END_VAR
END_METHOD

{attribute 'TcTypeSystem'}

METHOD FB_init : BOOL
VAR_INPUT
	bInitRetains : BOOL;
	bInCopyCode : BOOL;
END_VAR
END_METHOD

{attribute 'TcTypeSystem'}

{attribute 'monitoring' := 'call'}
	PROPERTY nHResult : HRESULT
GET
END_GET
END_PROPERTY

{attribute 'TcTypeSystem'}

{attribute 'monitoring' := 'call'}
	PROPERTY eInitExceptionHandling : E_FpExcptCtrlSetEx
GET
END_GET
SET
END_SET
END_PROPERTY

{attribute 'TcTypeSystem'}

{attribute 'monitoring' := 'call'}
	PROPERTY eUpdateExceptionHandling : E_FpExcptCtrlSetEx
GET
END_GET
SET
END_SET
END_PROPERTY

{attribute 'TcTypeSystem'}

{attribute 'monitoring' := 'call'}
	PROPERTY nExceptionCnt : ULINT
GET
END_GET
END_PROPERTY

{attribute 'TcTypeSystem'}

{attribute 'monitoring' := 'variable'}
	PROPERTY stActiveException : ST_ExceptionInfo
GET
END_GET
END_PROPERTY

{attribute 'TcTypeSystem'}

{attribute 'monitoring' := 'call'}
	PROPERTY bInitialized : BOOL
GET
END_GET
END_PROPERTY

{attribute 'TcTypeSystem'}

{attribute 'monitoring' := 'call'}
	PROPERTY bExecute : BOOL
GET
END_GET
SET
END_SET
END_PROPERTY

END_FUNCTION_BLOCK

// POUs/TcCOM Wrapper/FB_Copy_of_Sensor_model_new_TcCOM_InitStruct

{attribute 'c++_compatible'}
{attribute 'external_name' := 'FB_Copy_of_Sensor_model_new_TcCOM_InitStruct_GUID_FD0BCB26_D17A_EE83_BDA4_4D27D413E2A8'}
{attribute 'TcIecLibraryType'}
{attribute 'call_after_init'}
{attribute 'reflection'}
FUNCTION_BLOCK FB_Copy_of_Sensor_model_new_TcCOM_InitStruct
VAR
	{attribute 'hide'}
	{attribute 'no_copy'}
	{attribute 'GUID' := '18071995-0000-0000-0000-000000000018'}
	m_pData : PVOID;
	{attribute 'TcInitSymbol'}
	{attribute 'GUID' := '8007AE3B-86BB-40F2-B385-EF87FCC239A4'}
	eTraceLevelMaxFB : TcTraceLevel := TcTraceLevel.tlInfo;
	 {attribute 'hide'}
	_reserved1 : UDINT;
	{attribute 'hide'}
	{attribute 'instance-path'}
	{attribute 'noinit'}
	{attribute 'GUID' := '18071995-0000-0000-0000-0001000000FF'}
	sInstancePath : STRING(255);
	{attribute 'hide'}
	{attribute 'noinit'}
	{attribute 'GUID' := '18071995-0000-0000-0000-000000000019'}
	m_HResultLog : HRESULT;
	{attribute 'hide'}
	{attribute 'noinit'}
	{attribute 'GUID' := '18071995-0000-0000-0000-000000000019'}
	m_HResult : HRESULT;
	 {attribute 'hide'}
	_reserved2 : UINT_0_32;
	 {attribute 'hide'}
	_reserved3 : ARRAY [1..12] OF UINT_8_16;
	 {attribute 'hide'}
	_reserved4 : ARRAY [1..12] OF USINT;
END_VAR
VAR_INPUT
	stCopy_of_Sensor_model_new_U : ST_Copy_of_Sensor_model_new_U_T;
END_VAR
VAR_OUTPUT
	stCopy_of_Sensor_model_new_Y : ST_Copy_of_Sensor_model_new_Y_T;
END_VAR
VAR
	{attribute 'hide'}
	{attribute 'GUID' := '63EB1589-B180-DF9B-D7A8-37EE56025269'}
	_ipCopy_of_Sensor_model_new : POINTER TO ITcCopy_of_Sensor_model_new;
	stInit : ST_FB_Copy_of_Sensor_model_new_TcCOM_InitStruct;
END_VAR

{attribute 'TcTypeSystem'}

METHOD FB_init : BOOL
VAR_INPUT
	bInitRetains : BOOL;
	bInCopyCode : BOOL;
	{attribute 'GUID' := '33981638-E858-EA6F-B1C3-33CC5D188F64'}
	stInit : REFERENCE TO ST_FB_Copy_of_Sensor_model_new_TcCOM_InitStruct;
END_VAR
END_METHOD

{attribute 'TcTypeSystem'}

{attribute 'call_after_init'}
METHOD FB_afterinit : BOOL
END_METHOD

{attribute 'TcTypeSystem'}

METHOD Reinit : BOOL
VAR_INPUT
	{attribute 'GUID' := '33981638-E858-EA6F-B1C3-33CC5D188F64'}
	stReInit : ST_FB_Copy_of_Sensor_model_new_TcCOM_InitStruct;
END_VAR
END_METHOD

{attribute 'TcTypeSystem'}

METHOD FB_exit : BOOL
VAR_INPUT
	bInCopyCode : BOOL;
END_VAR
END_METHOD

{attribute 'TcTypeSystem'}

	PROPERTY eObjectState : TCOM_STATE
GET
END_GET
SET
END_SET
END_PROPERTY

{attribute 'TcTypeSystem'}

{attribute 'monitoring' := 'call'}
	PROPERTY nHResult : HRESULT
GET
END_GET
END_PROPERTY

{attribute 'TcTypeSystem'}

	PROPERTY ipTcComObject : ITComObject
GET
END_GET
END_PROPERTY

{attribute 'TcTypeSystem'}

	PROPERTY ipADI : ITcADI
GET
END_GET
END_PROPERTY

{attribute 'TcTypeSystem'}

	PROPERTY nTaskOid : OTCID
GET
END_GET
SET
END_SET
END_PROPERTY

{attribute 'TcTypeSystem'}

	PROPERTY nTaskPriority : UDINT
GET
END_GET
END_PROPERTY

{attribute 'TcTypeSystem'}

	PROPERTY nTaskCycleTimeNs : UDINT
GET
END_GET
END_PROPERTY

{attribute 'TcTypeSystem'}

	PROPERTY nTaskPort : UINT
GET
END_GET
END_PROPERTY

{attribute 'TcTypeSystem'}

	PROPERTY nTaskSortOrder : UDINT
GET
END_GET
SET
END_SET
END_PROPERTY

{attribute 'TcTypeSystem'}

	PROPERTY eTraceLevelMax : TcTraceLevel
GET
END_GET
SET
END_SET
END_PROPERTY

{attribute 'TcTypeSystem'}

	PROPERTY eModuleCaller : E_ModuleCaller
GET
END_GET
SET
END_SET
END_PROPERTY

{attribute 'TcTypeSystem'}

	PROPERTY eCallerVerification : E_CallerVerification
GET
END_GET
SET
END_SET
END_PROPERTY

{attribute 'TcTypeSystem'}

	PROPERTY eStepSizeAdaptation : E_StepSizeAdaptation
GET
END_GET
SET
END_SET
END_PROPERTY

{attribute 'TcTypeSystem'}

	PROPERTY eExecutionSequence : E_ExecutionSequence1
GET
END_GET
SET
END_SET
END_PROPERTY

{attribute 'TcTypeSystem'}

	PROPERTY bExecute : BOOL
GET
END_GET
SET
END_SET
END_PROPERTY

{attribute 'TcTypeSystem'}

	PROPERTY eAccessLockState : TCOM_STATE
GET
END_GET
SET
END_SET
END_PROPERTY

{attribute 'TcTypeSystem'}

	PROPERTY eInitExceptionHandling : E_FpExcptCtrlSet
GET
END_GET
SET
END_SET
END_PROPERTY

{attribute 'TcTypeSystem'}

	PROPERTY eUpdateExceptionHandling : E_FpExcptCtrlSetEx
GET
END_GET
SET
END_SET
END_PROPERTY

{attribute 'TcTypeSystem'}

	PROPERTY stModuleBuildInfo : ST_ModuleBuildInfo
GET
END_GET
END_PROPERTY

{attribute 'TcTypeSystem'}

	PROPERTY bInitialized : BOOL
GET
END_GET
END_PROPERTY

{attribute 'TcTypeSystem'}

	PROPERTY nSkippedExecutionCount : UDINT
GET
END_GET
END_PROPERTY

{attribute 'TcTypeSystem'}

	PROPERTY stLibraryInfo : ST_LibraryInfo
GET
END_GET
END_PROPERTY

{attribute 'TcTypeSystem'}

	PROPERTY stModuleInfo : ST_ModuleInfo
GET
END_GET
END_PROPERTY

{attribute 'TcTypeSystem'}

	PROPERTY stModuleGeneratorInfo : ST_TcMatSim_ModuleGeneratorInfo
GET
END_GET
SET
END_SET
END_PROPERTY

{attribute 'TcTypeSystem'}

	PROPERTY stSimulinkModelInfo : ST_TcMatSim_SimulinkModelInfo
GET
END_GET
SET
END_SET
END_PROPERTY

{attribute 'TcTypeSystem'}

	PROPERTY eCopy_of_Sensor_model_new_P_Sharing : E_ParameterSharingType
GET
END_GET
SET
END_SET
END_PROPERTY

{attribute 'TcTypeSystem'}

	PROPERTY nCopy_of_Sensor_model_new_P_Definer : OTCID
GET
END_GET
END_PROPERTY

{attribute 'TcTypeSystem'}

	PROPERTY stCopy_of_Sensor_model_new_P : ST_P_Copy_of_Sensor_model_new_T
GET
END_GET
SET
END_SET
END_PROPERTY

{attribute 'TcTypeSystem'}

	PROPERTY fSimulationTime : LREAL
GET
END_GET
END_PROPERTY

{attribute 'TcTypeSystem'}

	PROPERTY nCycleCount : ULINT
GET
END_GET
END_PROPERTY

{attribute 'TcTypeSystem'}

	PROPERTY nExceptionCount : ULINT
GET
END_GET
END_PROPERTY

{attribute 'TcTypeSystem'}

	PROPERTY stExceptionInfo : ST_ExceptionInfo
GET
END_GET
END_PROPERTY

END_FUNCTION_BLOCK
